# B&R Automation Studio project laba1KRBO0121
Automation Studio 4.5.2.102

## Configuration Config1

CPU 4PP065.0571-P74, AutomationRuntime D4.52, Build 4.1.2, Vc V4.52.0, Safety 1.6

### Task classes (Cpu.sw)
```
Cyclic#6:
  Program1 <- Program1.prg
Cyclic#7:
  Program2 <- Program2.prg
NcDataObjects: acp10etxen <- acp10etxen.dob, gAxis01a <- gAxis01obj.gAxis01a.dob, gAxis01i <- gAxis01obj.gAxis01i.dob, gAxis02a <- gAxis02obj.gAxis02a.dob, gAxis02i <- gAxis02obj.gAxis02i.dob
Binaries: TCData, udbdef, ashwd, Role, User, sysconf, ashwac, asfw, arconfig, iomap, Acp10map, acp10cfg
Libraries: Acp10man, Acp10par, NcGlobal, Acp10sdc, Acp10_MC, brsystem, sys_lib, runtime, AsBrStr, astime, fileio, powerlnk, asieccon
```

### Hardware
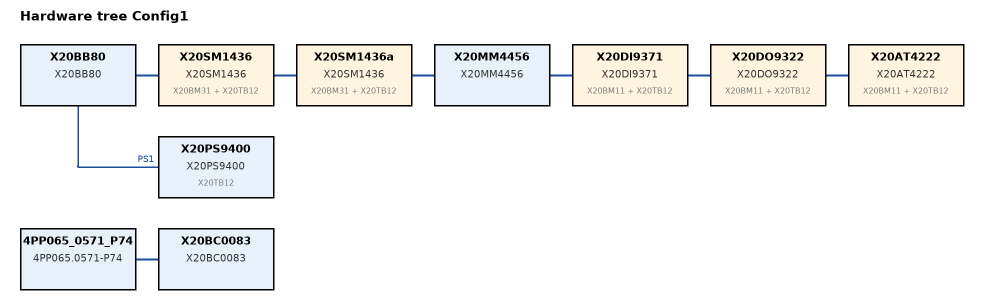
```
4PP065_0571_P74 : 4PP065.0571-P74 v1.1.2.0
  Connector IF4:
    Baudrate = 0
    InaNodeNumber = 1
  Connector IF5:
    ActivateDevice = 1
    Mode = Manual
    InternetAddress = 10.0.1.10
    SubnetMask = 255.255.255.0
  ConfigurationID = labBR
  TimerDeviceType = EPLX2X
  TimerDevice = 4PP065_0571_P74.IF4
  TaskClassIdleTime = 2000
  Cyclic1Duration = 2000
  Cyclic1Tolerance = 0
  Cyclic1Output = 1
X20AT4222 : X20AT4222 v1.2.3.0  [SS1 -> X20TB12e.SS; SL -> X20BM11b.SL1]
X20BB80 : X20BB80 v1.0.2.0
X20BC0083 : X20BC0083 v2.9.0.0  [PLK1 -> 4PP065_0571_P74.IF4 (NodeNumber=2) [Cable Type=PowerlinkCable, Length=10, Version=1.0.0.2]; SL -> X20BB80.SL1]
X20BM11 : X20BM11 v1.0.0.1  [X2X1 -> X20MM4456.X2X2]
X20BM11a : X20BM11 v1.0.0.1  [X2X1 -> X20BM11.X2X2]
X20BM11b : X20BM11 v1.0.0.1  [X2X1 -> X20BM11a.X2X2]
X20BM31 : X20BM31 v1.0.0.1  [X2X1 -> X20BB80.IF1]
X20BM31a : X20BM31 v1.0.0.1  [X2X1 -> X20BM31.X2X2]
X20DI9371 : X20DI9371 v1.0.2.0  [SS1 -> X20TB12c.SS; SL -> X20BM11.SL1]
X20DO9322 : X20DO9322 v1.0.3.0  [SS1 -> X20TB12d.SS; SL -> X20BM11a.SL1]
X20MM4456 : X20MM4456 v1.1.5.0  [X2X1 -> X20BM31a.X2X2]
X20PS9400 : X20PS9400 v1.0.2.4  [SS1 -> X20TB12.SS; PS -> X20BB80.PS1]
X20SM1436 : X20SM1436 v1.4.2.1  [SS1 -> X20TB12a.SS; SL -> X20BM31.SL1]
X20SM1436a : X20SM1436 v1.4.2.1  [SS1 -> X20TB12b.SS; SL -> X20BM31a.SL1]
X20TB12 : X20TB12 v1.0.0.0
X20TB12a : X20TB12 v1.0.0.0
X20TB12b : X20TB12 v1.0.0.0
X20TB12c : X20TB12 v1.0.0.0
X20TB12d : X20TB12 v1.0.0.0
X20TB12e : X20TB12 v1.0.0.0
```

### IoMap.iom - 4PP065_0571_P74/IoMap.iom
```iecst
VAR_CONFIG
	Cyclic#1.gAxis01_DrvIf.iLifeCnt AT %IB."X20SM1436".LifeCnt;
	Cyclic#1.gAxis01_DrvIf.iDrvOK AT %IX."X20SM1436".DrvOk01;
	Cyclic#1.gAxis01_DrvIf.oBoostCurrent AT %QX."X20SM1436".BoostCurrent01;
	Cyclic#1.gAxis01_DrvIf.oStandStillCurrent AT %QX."X20SM1436".StandstillCurrent01;
	Cyclic#1.gAxis01_DrvIf.oSetTime AT %QW."X20SM1436".SetTime01;
	Cyclic#1.gAxis01_MotorStep0 AT %QW."X20SM1436".Motor1Step0;
	Cyclic#1.gAxis01_DiDoIf.iLifeCntDriveEnable AT %IB."X20SM1436".LifeCnt;
	Cyclic#1.gAxis01_DiDoIf.iLifeCntDriveReady AT %IB."X20SM1436".LifeCnt;
	Cyclic#1.gAxis01_DiDoIf.iDriveReady AT %IX."X20SM1436".DrvOk01;
	Cyclic#1.gAxis01_DiDoIf.oDriveEnable AT %QX."X20SM1436".DriveEnable01;
	Cyclic#1.gAxis01_EncIf1.iLifeCnt AT %IB."X20SM1436".LifeCnt;
	Cyclic#1.gAxis01_EncIf1.iEncOK AT %IX."X20SM1436".EncOk01;
	Cyclic#1.gAxis01_EncIf1.iActPos AT %IW."X20SM1436".ActPos01;
	Cyclic#1.gAxis01_EncIf1.iRefPulsePos AT %IW."X20SM1436".RefPulsePos01;
	Cyclic#1.gAxis01_EncIf1.iRefPulseCnt AT %IB."X20SM1436".RefPulseCnt01;
	Cyclic#1.gAxis01_EncIf1.iActTime AT %IW."X20SM1436".ActTime01;
	Cyclic#1.gAxis02_DrvIf.iLifeCnt AT %IB."X20SM1436a".LifeCnt;
	Cyclic#1.gAxis02_DrvIf.iDrvOK AT %IX."X20SM1436a".DrvOk01;
	Cyclic#1.gAxis02_DrvIf.oBoostCurrent AT %QX."X20SM1436a".BoostCurrent01;
	Cyclic#1.gAxis02_DrvIf.oStandStillCurrent AT %QX."X20SM1436a".StandstillCurrent01;
	Cyclic#1.gAxis02_DrvIf.oSetTime AT %QW."X20SM1436a".SetTime01;
	Cyclic#1.gAxis02_MotorStep0 AT %QW."X20SM1436a".Motor1Step0;
	Cyclic#1.gAxis02_DiDoIf.iLifeCntDriveEnable AT %IB."X20SM1436a".LifeCnt;
	Cyclic#1.gAxis02_DiDoIf.iLifeCntDriveReady AT %IB."X20SM1436a".LifeCnt;
	Cyclic#1.gAxis02_DiDoIf.iDriveReady AT %IX."X20SM1436a".DrvOk01;
	Cyclic#1.gAxis02_DiDoIf.oDriveEnable AT %QX."X20SM1436a".DriveEnable01;
	Cyclic#1.gAxis02_EncIf1.iLifeCnt AT %IB."X20SM1436a".LifeCnt;
	Cyclic#1.gAxis02_EncIf1.iEncOK AT %IX."X20SM1436a".EncOk01;
	Cyclic#1.gAxis02_EncIf1.iActPos AT %IW."X20SM1436a".ActPos01;
	Cyclic#1.gAxis02_EncIf1.iRefPulsePos AT %IW."X20SM1436a".RefPulsePos01;
	Cyclic#1.gAxis02_EncIf1.iRefPulseCnt AT %IB."X20SM1436a".RefPulseCnt01;
	Cyclic#1.gAxis02_EncIf1.iActTime AT %IW."X20SM1436a".ActTime01;
	::Program1:Led_1 AT %QX."X20DO9322".DigitalOutput02;
	::Program2:Led_2 AT %QX."X20DO9322".DigitalOutput03;
END_VAR
```

## Logical view

### Global.var - Global variables
```iecst
VAR
	gAxis01 : ACP10AXIS_typ;
	gAxis01_HW : SdcHwCfg_typ := (0);
	gAxis01_DrvIf : SdcDrvIf16_typ := (0);
	gAxis01_EncIf1 : SdcEncIf16_typ := (0);
	gAxis01_DiDoIf : SdcDiDoIf_typ := (0);
	gAxis01_MotorStep0 : INT := (0);
	gAxis02 : ACP10AXIS_typ;
	gAxis02_HW : SdcHwCfg_typ := (0);
	gAxis02_DrvIf : SdcDrvIf16_typ := (0);
	gAxis02_EncIf1 : SdcEncIf16_typ := (0);
	gAxis02_DiDoIf : SdcDiDoIf_typ := (0);
	gAxis02_MotorStep0 : INT := (0);
END_VAR
```

### Program Logical/Program2 (ANSIC)

#### Variables.var
```iecst
VAR
	Led_2 : BOOL;
END_VAR
```

#### Main.c
```c
#include <bur/plctypes.h>

#ifdef _DEFAULT_INCLUDES
	#include <AsDefault.h>
#endif

void _INIT ProgramInit(void)
{
	Led_2 = 0;
}

void _CYCLIC ProgramCyclic(void)
{
	if (Led_2 == 0)
	{
		Led_2 = 1;
	}
	else
	{
		Led_2 = 0;
	}
}

void _EXIT ProgramExit(void)
{

}
```

### Program Logical/Program1 (ANSIC)

#### Variables.var
```iecst
VAR
	Led_1 : BOOL;
END_VAR
```

#### Main.c
```c
#include <bur/plctypes.h>

#ifdef _DEFAULT_INCLUDES
	#include <AsDefault.h>
#endif

void _INIT ProgramInit(void)
{
	Led_1 = 0;
}

void _CYCLIC ProgramCyclic(void)
{
	if (Led_1 == 0)
	{
		Led_1 = 1;
	}
	else
	{
		Led_1 = 0;
	}
}

void _EXIT ProgramExit(void)
{

}
```

Listed in the project but not available here: Logical/Global.typ, Logical/Libraries, Logical/ncsdcctrl, Logical/acp10etxen, Logical/gAxis01obj, Logical/gAxis02obj
